(* CoDeSys 2.3 export: TUZSPEED.EXP *)

(* Data type *)
TYPE tUZSpeed : REAL;
END_TYPE
